// Mitsubishi GX Works2 project: 2023-05-26 #1 생산자동화기능사 18번   PLC: Q03UDV
// 생산자동화기능사

// global labels: Global1
VAR_GLOBAL
  PB1 AT X0 : BOOL;
  PB2 AT X1 : BOOL;
  정지 AT X2 : BOOL;
  공급후진 AT X3 : BOOL;
  공급전진 AT X4 : BOOL;
  가공후진 AT X5 : BOOL;
  가공전진 AT X6 : BOOL;
  송출후진 AT X7 : BOOL;
  송출전진 AT X8 : BOOL;
  배출후진 AT X9 : BOOL;
  배출전진 AT X0A : BOOL;
  매거진 AT X0B : BOOL;
  금속센서 AT X0F : BOOL;
  PB3 AT X0C : BOOL;
  적색 AT Y20 : BOOL;
  황색 AT Y21 : BOOL;
  녹색 AT Y22 : BOOL;
  공급1 AT Y23 : BOOL;
  공급2 AT Y24 : BOOL;
  가공 AT Y25 : BOOL;
  드릴 AT Y26 : BOOL;
  송출 AT Y27 : BOOL;
  배출 AT Y28 : BOOL;
  컨베이어 AT Y29 : BOOL;
END_VAR

PROGRAM 테스트동작
VAR
  STATE : INT;
END_VAR
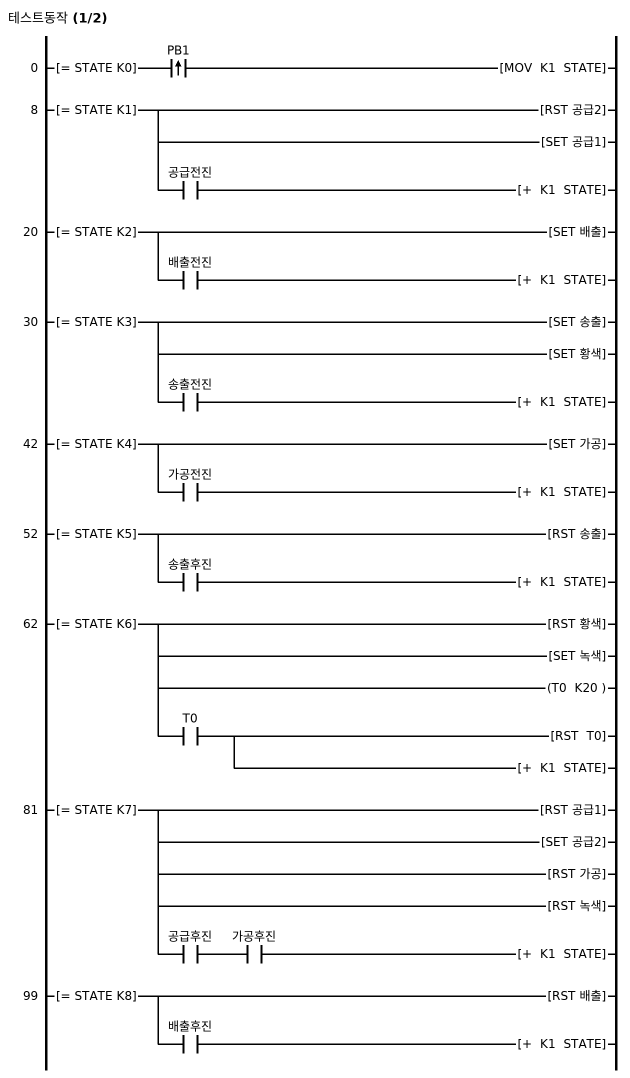
0     LD=     STATE K0
      ANDP    PB1
      MOV     K1 STATE
8     LD=     STATE K1
      RST     공급2
      SET     공급1
      AND     공급전진
      +       K1 STATE
20    LD=     STATE K2
      SET     배출
      AND     배출전진
      +       K1 STATE
30    LD=     STATE K3
      SET     송출
      SET     황색
      AND     송출전진
      +       K1 STATE
42    LD=     STATE K4
      SET     가공
      AND     가공전진
      +       K1 STATE
52    LD=     STATE K5
      RST     송출
      AND     송출후진
      +       K1 STATE
62    LD=     STATE K6
      RST     황색
      SET     녹색
      OUT     T0 K20
      AND     T0
      RST     T0
      +       K1 STATE
81    LD=     STATE K7
      RST     공급1
      SET     공급2
      RST     가공
      RST     녹색
      AND     공급후진
      AND     가공후진
      +       K1 STATE
99    LD=     STATE K8
      RST     배출
      AND     배출후진
      +       K1 STATE
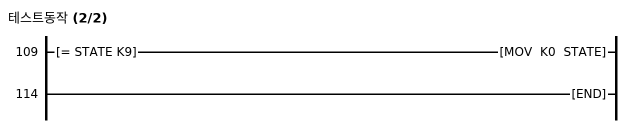
109   LD=     STATE K9
      MOV     K0 STATE
114   END
END_PROGRAM

PROGRAM 단속연속동작
VAR
  STATE : INT;
  MODE : INT;
END_VAR
VAR CONSTANT
  단속 : INT;
  연속 : INT := 1;
END_VAR
VAR
  CNT_비금속 : ;
  CNT_금속 : ;
END_VAR
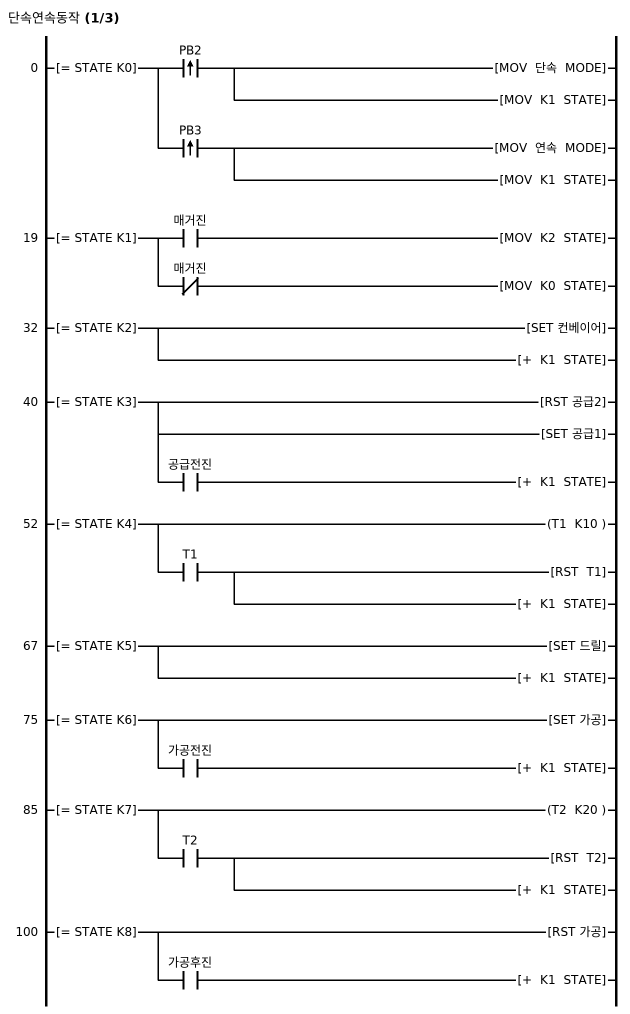
0     LD=     STATE K0
      MPS
      ANDP    PB2
      MOV     단속 MODE
      MOV     K1 STATE
      MPP
      ANDP    PB3
      MOV     연속 MODE
      MOV     K1 STATE
19    LD=     STATE K1
      MPS
      AND     매거진
      MOV     K2 STATE
      MPP
      ANI     매거진
      MOV     K0 STATE
32    LD=     STATE K2
      SET     컨베이어
      +       K1 STATE
40    LD=     STATE K3
      RST     공급2
      SET     공급1
      AND     공급전진
      +       K1 STATE
52    LD=     STATE K4
      OUT     T1 K10
      AND     T1
      RST     T1
      +       K1 STATE
67    LD=     STATE K5
      SET     드릴
      +       K1 STATE
75    LD=     STATE K6
      SET     가공
      AND     가공전진
      +       K1 STATE
85    LD=     STATE K7
      OUT     T2 K20
      AND     T2
      RST     T2
      +       K1 STATE
100   LD=     STATE K8
      RST     가공
      AND     가공후진
      +       K1 STATE
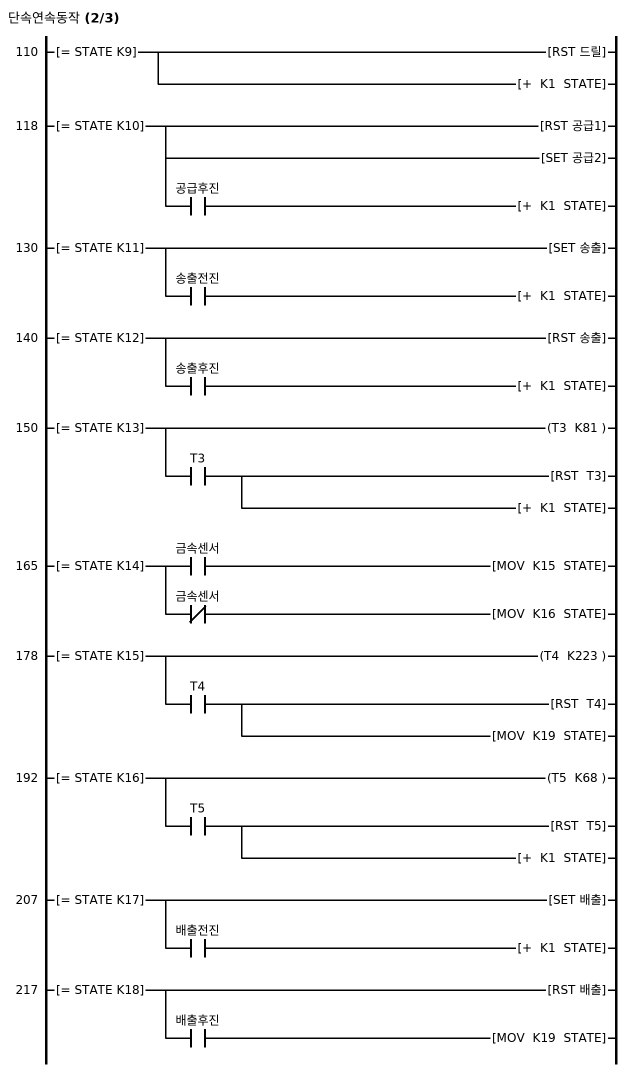
110   LD=     STATE K9
      RST     드릴
      +       K1 STATE
118   LD=     STATE K10
      RST     공급1
      SET     공급2
      AND     공급후진
      +       K1 STATE
130   LD=     STATE K11
      SET     송출
      AND     송출전진
      +       K1 STATE
140   LD=     STATE K12
      RST     송출
      AND     송출후진
      +       K1 STATE
150   LD=     STATE K13
      OUT     T3 K81
      AND     T3
      RST     T3
      +       K1 STATE
165   LD=     STATE K14
      MPS
      AND     금속센서
      MOV     K15 STATE
      MPP
      ANI     금속센서
      MOV     K16 STATE
178   LD=     STATE K15
      OUT     T4 K223
      AND     T4
      RST     T4
      MOV     K19 STATE
192   LD=     STATE K16
      OUT     T5 K68
      AND     T5
      RST     T5
      +       K1 STATE
207   LD=     STATE K17
      SET     배출
      AND     배출전진
      +       K1 STATE
217   LD=     STATE K18
      RST     배출
      AND     배출후진
      MOV     K19 STATE
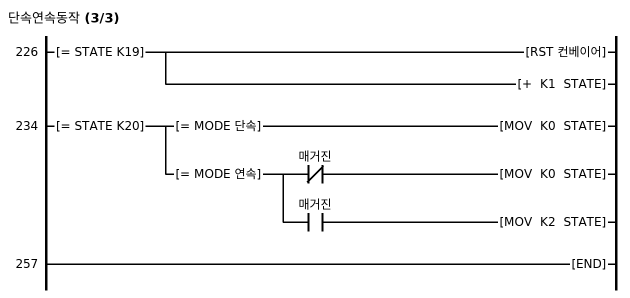
226   LD=     STATE K19
      RST     컨베이어
      +       K1 STATE
234   LD=     STATE K20
      MPS
      AND=    MODE 단속
      MOV     K0 STATE
      MPP
      AND=    MODE 연속
      MPS
      ANI     매거진
      MOV     K0 STATE
      MPP
      AND     매거진
      MOV     K2 STATE
257   END
END_PROGRAM
